Universal Robots PolyScope program: send_currrent_pose_to_socket.urp

Program send_currrent_pose_to_socket (installation=default directory=/home/ur/ursim-current/programs createdIn=3.11.0.82155 lastSavedIn=3.11.0.82155 robotSerialNumber=20183599999)
Calibrated DH parameters: a=[0, -0.425, -0.39225, 0, 0, 0]; d=[0.089159, 0, 0, 0.10915, 0.09465, 0.0823]; alpha=[1.570796, 0, 0, 1.570796, -1.570796, 0]; deltaTheta=[0, 0, 0, 0, 0, 0]
BeforeStart
  host := "10.8.8.200"
  port := 30002
  socket := False
  socket_name := "socket_0"
  socket_send := False
Robot Program (runOnlyOnce=true)
  Loop While (checkContinuously=false) expression=socket≠ True
    socket := socket_open(host, port, socket_name)
    Wait Sleep waitTime=1
  current_pose := get_actual_tcp_pose()
  Loop While (checkContinuously=false) expression=socket_send≠ True
    SuppressedNode
      socket_send := socket_send_int(current_pose, "socket_0")
    socket_send := socket_send_string(current_pose, "socket_0")
    Wait Sleep waitTime=1
  socket_send := False
  Script: socket_close(socket_name)
  socket := False
